				IF TriggerInput.Mode = TOUCHPROBEMODE_SINGLE_COMPATIBILITYMODE THEN
					CASE TriggerInput.Edge OF
						RisingEdge :
							IndexOffset := 16#201;
						FallingEdge:
							IndexOffset := 16#202;
					ELSE (* case *)
						Error := TRUE;
						ErrorID := MC_ERROR_INVALID_TOUCH_PROBE;
					END_CASE
				ELSE
					IF TcMcGlobal.NcDeviceInfoNcVersion > 16#020B07DD THEN
						IndexOffset := 16#200;  (* new from 2.11 NC driver 2014 *)
					ELSE
						(* new probe mode with old NC driver not possible *)
						Error := TRUE;
						ErrorID := MC_ERROR_INVALID_TOUCH_PROBE;
					END_IF
				END_IF

				IF TriggerInput.EncoderID > 255 THEN
					Error := TRUE;
					ErrorID := MC_ERROR_INVALID_TOUCH_PROBE;
				END_IF

				IF NOT Error THEN
					CASE TriggerInput.TouchProbe OF
						TouchProbe1,
						TouchProbe2,
						TouchProbe3,
						TouchProbe4:
							(* activate latch *)
							iTriggerInput := TriggerInput; (* save local copy *)
							ActTouchProbeActivate();
							iState := STATE_ORDER;

						PlcEvent:
							(* no action necessary here *);
							TriggerInput.ProbeState := TouchProbeActivated;
							iTriggerInput := TriggerInput; (* save local copy *)
							iState := STATE_WAITING;
					ELSE
						Error := TRUE;
						ErrorID := MC_ERROR_INVALID_TOUCH_PROBE;
					END_CASE
				END_IF
			END_IF
		END_IF

	STATE_ORDER :	(* wait until probe is activated *)
		ActTouchProbeActivate();

	STATE_WAITING : (* wait until touch probe was trigerred *)
		CASE iTriggerInput.TouchProbe OF (* type of touch probe *)
			TouchProbe1,
			TouchProbe2,
			TouchProbe3,
			TouchProbe4:
				IF TcMcGlobal.NcDeviceInfoNcVersion > 16#020B07DD AND stTouchProbeActivation.Mode<>INT_TO_UDINT(TOUCHPROBEMODE_SINGLE_COMPATIBILITYMODE) THEN
					(* new touch probe interface since TwinCAT 2.11 Nc-Driver 2014 *)
					ActTouchProbeMonitoring();
				ELSE
					(* classic touch probe interface until TwinCAT 2.11 Nc-Driver 2013 *)
					ActTouchProbeMonitorLatchValid();
					IF iState=STATE_WAITING THEN (* still not triggered *)
						ActTouchProbeMonitorActivity();
					END_IF
				END_IF

			(* CASE PlcEvent *)
			PlcEvent : (* touch proble will be triggered through a PLC signal (iTriggerInput.PlcEvent) *)
				ActTouchProbeMonitorPlcEvent();
		END_CASE (* type of touch probe *)

		IF NOT Done AND (TriggerInput.ProbeState = TouchProbeAborted) THEN
			(* function block has been aborted by an external MC_AbortTrigger *)
			CommandAborted := TRUE;
			iState := STATE_INITIALIZATION;
		END_IF

		IF TriggerInput.Mode = TOUCHPROBEMODE_CONTINOUS THEN
			(* check if probe triggered, then restart probe *)
			IF Done AND Execute THEN
(*				fbAdsReadState(READ:=FALSE); *)
(*				LastTouchProbeValue := TouchProbeValue;
				LastTouchProbeCounter := TouchProbeCounter;
				fbAdsReadLatchStatus(WRTRD:=TRUE); *)(* retrigger *)
				iState := STATE_WAITING; (* keep on waiting for next trigger *)
			ELSIF NOT Execute THEN (* abort trigger *)
				stTouchProbeDeactivation.TouchProbe := iTriggerInput.TouchProbe;
				stTouchProbeDeactivation.Edge := iTriggerInput.Edge;
				fbADSwrite(	WRITE:=FALSE); (* reset *)
				fbADSwrite(	NETID:= TcMcGlobal.NCNETID_TCMC,
							PORT:=AMSPORT_R0_NCSAF ,
							IDXGRP:=16#5200+TriggerInput.EncoderID ,
							IDXOFFS:=16#205,	(* deactivate touch probe *)
							LEN:= SIZEOF(stTouchProbeDeactivation),
							SRCADDR:=ADR(stTouchProbeDeactivation),
							WRITE:=TRUE ,
							TMOUT:=TcMcGlobal.tADSTimeOut);
				iState := 30000;
			END_IF
		END_IF

		IF iState<> STATE_WAITING THEN
			(* leave the waiting state now *)
			TriggerInput.ProbeState := TouchProbeInactive;
			fbAdsReadModulo(READ:=FALSE);	(* initialize again during next cycle *)
		END_IF

	30000 : (* abort trigger *)
		fbADSwrite();
		IF NOT fbAdsWrite.BUSY THEN
			IF fbAdsWrite.ERR THEN
				Error := fbAdsWrite.ERR;
				ErrorID := fbAdsWrite.ERRID;
			END_IF
			iState := STATE_INITIALIZATION;
		END_IF

END_CASE

ADSbusy := fbAdsWrite.BUSY OR fbAdsReadValid.BUSY OR fbAdsReadValue.BUSY OR fbAdsReadState.BUSY OR fbAdsReadModulo.BUSY;
IF iState=STATE_INITIALIZATION AND NOT Restart THEN
	(* reset Busy immediately  when sequence ends *)
	Busy := FALSE;
END_IF
END_FUNCTION_BLOCK
ACTION ActTouchProbeActivate:
(* start the touch probe sequence *)

(*LatchID := iTriggerInput.TouchProbe;*)
TriggerInput.ProbeState := TouchProbeActivated;
iTriggerInput.ProbeState := TouchProbeActivated;

(* read version of NC *)
(*
IF TcMcGlobal.NcDeviceInfoNcVersion=0 THEN
	TcMcGlobal.ReadDeviceInfo();
END_IF
*)

stTouchProbeActivation.TouchProbe := iTriggerInput.TouchProbe;
stTouchProbeActivation.Edge := iTriggerInput.Edge;
stTouchProbeActivation.Mode := iTriggerInput.Mode;
stTouchProbeActivation.SignalSource := iTriggerInput.SignalSource;	(* 20110218 KSt *)

IF stTouchProbeActivation.Mode = INT_TO_UDINT(TOUCHPROBEMODE_SINGLE_COMPATIBILITYMODE) THEN
	fbADSwrite(	NETID:= TcMcGlobal.NCNETID_TCMC,
				PORT:=AMSPORT_R0_NCSAF ,
				IDXGRP:=16#5200+iTriggerInput.EncoderID ,
				IDXOFFS:=IndexOffset,
				LEN:=0,
				SRCADDR:=ADR(stTouchProbeActivation),
				WRITE:=TRUE ,
				TMOUT:=TcMcGlobal.tADSTimeOut);
ELSE
	fbADSwrite(	NETID:= TcMcGlobal.NCNETID_TCMC,
				PORT:=AMSPORT_R0_NCSAF ,
				IDXGRP:=16#5200+iTriggerInput.EncoderID ,
				IDXOFFS:=IndexOffset,
				LEN:=SIZEOF(stTouchProbeActivation),
				SRCADDR:=ADR(stTouchProbeActivation),
				WRITE:=TRUE ,
				TMOUT:=TcMcGlobal.tADSTimeOut);
END_IF

IF NOT fbADSwrite.BUSY THEN
	IF fbADSwrite.ERR THEN
		Error := fbADSwrite.ERR;
		ErrorID := fbADSwrite.ERRID;
	END_IF
	IF NOT Error AND iTriggerInput.ProbeState = TouchProbeAborted THEN
		(* Synchronization error between MC_TouchProbe and MC_AbortTrigger *)
		Error := TRUE;
		ErrorID := MC_ERROR_TOUCH_PROBE_DEACTIVATED;
	END_IF
	iTriggerInput.ProbeState := SEL( Error, TouchProbeActivated, TouchProbeInactive );
	iState := SEL( Error, STATE_WAITING, STATE_INITIALIZATION);
END_IF
END_ACTION
ACTION ActTouchProbeMonitorActivity:
(* check if latch is still active *)
TimerAdsReadState(IN := NOT TimerAdsReadState.q , PT:=T#1s);
IF TimerAdsReadState.q OR fbAdsReadState.BUSY THEN
	fbAdsReadState(	NETID:= TcMcGlobal.NCNETID_TCMC,
				PORT:=AMSPORT_R0_NCSAF ,
				IDXGRP:=16#5100+TriggerInput.EncoderID ,
				IDXOFFS:= 16#201,
				LEN:= SIZEOF(TouchProbeActive[1]),
				DESTADDR:=ADR(TouchProbeActive) ,
				READ:=TRUE ,
				TMOUT:=TcMcGlobal.tADSTimeOut );
	IF NOT fbAdsReadState.BUSY THEN
		IF fbAdsReadState.ERR THEN
			Error := TRUE;
			ErrorID := fbAdsReadState.ERRID;
		ELSE
			IF TouchProbeActive[TriggerInput.TouchProbe]<>1 THEN
				TouchProbeInactiveCounter[TriggerInput.TouchProbe] := TouchProbeInactiveCounter[TriggerInput.TouchProbe] + 1;
				IF TouchProbeInactiveCounter[TriggerInput.TouchProbe] > 1 THEN
					(* error condition when the probing sequence is inactive more than once *)
					Error := TRUE;
					ErrorID := MC_ERROR_TOUCH_PROBE_DEACTIVATED;
					CommandAborted := TRUE;
					iState := STATE_INITIALIZATION;
				END_IF
			END_IF
		END_IF
		fbAdsReadState(READ:=FALSE); (* reset *)
	END_IF
END_IF
END_ACTION
ACTION ActTouchProbeMonitoring:
(* 	monitor if the touch probe has been triggered and if it is still active *)

(* 	new touch probe interface since 4/2010
	This action is only used with the new interface 
*)

Done := FALSE;		(* default *)
RecordedPosition := 0;	(* default *)

(* check if latch is still active and check for valid latch *)
TimerAdsReadState(IN := NOT TimerAdsReadState.q , PT:=T#1s);
IF ExternalLatchValid OR TimerAdsReadState.q OR fbAdsReadLatchStatus.BUSY THEN
	(* request for this probe unit *)
	stTouchProbeStatusRequest.TouchProbe := iTriggerInput.TouchProbe;

	fbAdsReadLatchStatus(
		NETID:= TcMcGlobal.NCNETID_TCMC,
		PORT:=AMSPORT_R0_NCSAF ,
		IDXGRP:=16#5100+iTriggerInput.EncoderID ,
		IDXOFFS:= 16#200,
		WRITELEN:= SIZEOF(stTouchProbeStatusRequest),
		READLEN:= SIZEOF(stTouchProbeStatusResponse),
		SRCADDR:= ADR(stTouchProbeStatusRequest),
		DESTADDR:= ADR(stTouchProbeStatusResponse),
		WRTRD:= TRUE,
		TMOUT:= TcMcGlobal.tADSTimeOut );

	IF NOT fbAdsReadLatchStatus.BUSY THEN
		IF fbAdsReadLatchStatus.ERR THEN
			Error := TRUE;
			ErrorID := fbAdsReadLatchStatus.ERRID;
		ELSE
			IF iTriggerInput.Edge = FallingEdge THEN
				TouchProbeActive[iTriggerInput.TouchProbe] := stTouchProbeStatusResponse.FallingEdgeActive;
				TouchProbeValid[iTriggerInput.TouchProbe] := stTouchProbeStatusResponse.FallingEdgeValid;
				TouchProbeValue[iTriggerInput.TouchProbe] := stTouchProbeStatusResponse.FallingEdgeValue;
				TouchProbeCounter[iTriggerInput.TouchProbe] := stTouchProbeStatusResponse.FallingEdgeCounter;
			ELSE
				TouchProbeActive[iTriggerInput.TouchProbe] := stTouchProbeStatusResponse.RisingEdgeActive;
				TouchProbeValid[iTriggerInput.TouchProbe] := stTouchProbeStatusResponse.RisingEdgeValid;
				TouchProbeValue[iTriggerInput.TouchProbe] := stTouchProbeStatusResponse.RisingEdgeValue;
				TouchProbeCounter[iTriggerInput.TouchProbe] := stTouchProbeStatusResponse.RisingEdgeCounter;
			END_IF
			IF TouchProbeValid[iTriggerInput.TouchProbe] = 1 THEN
				IF  iTriggerInput.Mode <> TOUCHPROBEMODE_CONTINOUS		(* single mode *)
					OR LastTouchProbeValue[ iTriggerInput.TouchProbe ] <> TouchProbeValue[ iTriggerInput.TouchProbe ] 	(* or continous mode and value changed *)
					OR LastTouchProbeCounter[ iTriggerInput.TouchProbe ] <> TouchProbeCounter[ iTriggerInput.TouchProbe ](* or continous mode and counter changed *)
					THEN (* new position recorded  *)
					RecordedPosition:=TouchProbeValue[iTriggerInput.TouchProbe];
					LastTouchProbeValue := TouchProbeValue;
					LastTouchProbeCounter := TouchProbeCounter;
					Done := TRUE;
					IF TriggerInput.ModuloPositions AND (ModuloFactor<>0) THEN	(* check for  (ModuloFactor=0) - 2007-02-06 KSt *)
						RecordedPosition := MODABS(RecordedPosition,  ModuloFactor);
						TouchProbeModuloValue[TriggerInput.TouchProbe] := RecordedPosition;
(*						InWindow := (RecordedPosition>=FirstPosition) AND (RecordedPosition<=LastPosition);*)	(* 20110216 KSt *)
						IF FirstPosition>LastPosition THEN (* 20110216 KSt *)
							InWindow := (RecordedPosition>=FirstPosition) OR  (RecordedPosition<=LastPosition);  (* 20110216 KSt *)
						ELSE
							InWindow := (RecordedPosition>=FirstPosition) AND (RecordedPosition<=LastPosition);
						END_IF
					ELSE
						InWindow := (RecordedPosition>=FirstPosition) AND (RecordedPosition<=LastPosition);
					END_IF
					IF WindowOnly AND NOT InWindow THEN
						RecordedPosition:=0;
						Done := FALSE;
						Restart := TRUE; (* ignore this event, latch next one *)
					ELSE
						(* fill RecordedData structure *)
						RecordedData.RecordedPosition := RecordedPosition;
						RecordedData.Counter:=TouchProbeCounter[TriggerInput.TouchProbe];
						RecordedData.AbsolutePosition := TouchProbeValue[iTriggerInput.TouchProbe];
						IF ModuloFactor = 0 THEN
							RecordedData.ModuloPosition := MODABS(RecordedData.AbsolutePosition,  360);
						ELSE
							RecordedData.ModuloPosition := MODABS(RecordedData.AbsolutePosition,  ModuloFactor);
						END_IF
					END_IF
					iState := STATE_INITIALIZATION;
				END_IF
			ELSIF TouchProbeActive[iTriggerInput.TouchProbe] <> 1 THEN
				TouchProbeInactiveCounter[iTriggerInput.TouchProbe] := TouchProbeInactiveCounter[iTriggerInput.TouchProbe] + 1;
				IF TouchProbeInactiveCounter[iTriggerInput.TouchProbe] > 1 THEN
					(* error condition when the probing sequence is inactive more than once *)
					Error := TRUE;
					ErrorID := MC_ERROR_TOUCH_PROBE_DEACTIVATED;
					CommandAborted := TRUE;
					iState := STATE_INITIALIZATION;
				END_IF
			END_IF
		END_IF
		fbAdsReadLatchStatus(WRTRD:=FALSE); (* reset *)
		IF iTriggerInput.Mode=TOUCHPROBEMODE_CONTINOUS AND Execute THEN
			fbAdsReadLatchStatus(WRTRD:=TRUE); (* retrigger *)
		END_IF
	END_IF
END_IF
END_ACTION
ACTION ActTouchProbeMonitorLatchValid:
(* monitor if the touch probe has been triggered *)

IF F_AxisExternalLatchValid(Axis.NcToPlc.StateDWord) THEN
	(* read the status of the latch *)
	fbAdsReadValid(	NETID:= TcMcGlobal.NCNETID_TCMC,
				PORT:=AMSPORT_R0_NCSAF ,
				IDXGRP:=16#5100+TriggerInput.EncoderID ,
				IDXOFFS:= 16#202,
				LEN:= SIZEOF(TouchProbeValid[1]),
				DESTADDR:=ADR(TouchProbeValid) ,
				READ:=TRUE ,
				TMOUT:=TcMcGlobal.tADSTimeOut );
	(* read the latched value *)
	fbAdsReadValue(	NETID:= TcMcGlobal.NCNETID_TCMC,
				PORT:=AMSPORT_R0_NCSAF ,
				IDXGRP:=16#5100+TriggerInput.EncoderID ,
				IDXOFFS:= 16#205,
				LEN:=SIZEOF(TouchProbeValue[1]),
				DESTADDR:=ADR(TouchProbeValue) ,
				READ:=TRUE ,
				TMOUT:=TcMcGlobal.tADSTimeOut );
	IF NOT fbAdsReadValid.BUSY AND NOT fbAdsReadValue.BUSY THEN
		IF fbAdsReadValid.err THEN
			Error := TRUE;
			ErrorID := fbAdsReadValid.ERRID;
			iState := STATE_INITIALIZATION;
		ELSIF fbAdsReadValue.err THEN
			Error := TRUE;
			ErrorID := fbAdsReadValue.ERRID;
			iState := STATE_INITIALIZATION;
		ELSE (* no error *)
			IF TouchProbeValid[TriggerInput.TouchProbe]=1 THEN
				RecordedPosition:=TouchProbeValue[TriggerInput.TouchProbe];
				Done := TRUE;
				IF TriggerInput.ModuloPositions AND (ModuloFactor<>0) THEN	(* check for  (ModuloFactor=0) - 2007-02-06 KSt *)
					RecordedPosition := MODABS(RecordedPosition,  ModuloFactor);
					TouchProbeModuloValue[TriggerInput.TouchProbe] := RecordedPosition;
(*					InWindow := (RecordedPosition>=FirstPosition) AND (RecordedPosition<=LastPosition);*)  (* 20110216 KSt *)
					IF FirstPosition>LastPosition THEN (* 20110216 KSt *)
						InWindow := (RecordedPosition>=FirstPosition) OR  (RecordedPosition<=LastPosition);  (* 20110216 KSt *)
					ELSE
						InWindow := (RecordedPosition>=FirstPosition) AND (RecordedPosition<=LastPosition);
					END_IF
				ELSE
					InWindow := (RecordedPosition>=FirstPosition) AND (RecordedPosition<=LastPosition);
				END_IF
				IF WindowOnly AND NOT InWindow THEN
					RecordedPosition:=0;
					Done := FALSE;
					Restart := TRUE; (* ignore this event, latch next one *)
				ELSE
					(* fill RecordedData structure *)
					RecordedData.RecordedPosition := RecordedPosition;
					RecordedData.Counter:=TouchProbeCounter[TriggerInput.TouchProbe];
					RecordedData.AbsolutePosition := TouchProbeValue[TriggerInput.TouchProbe];
					IF ModuloFactor = 0 THEN
						RecordedData.ModuloPosition := MODABS(RecordedData.AbsolutePosition,  360);
					ELSE
						RecordedData.ModuloPosition := MODABS(RecordedData.AbsolutePosition,  ModuloFactor);
					END_IF
				END_IF
				iState := STATE_INITIALIZATION;
			ELSE
				fbAdsReadValid(READ:=FALSE);
				fbAdsReadValue(READ:=FALSE);
			END_IF
		END_IF
	END_IF
END_IF
END_ACTION
ACTION ActTouchProbeMonitorPlcEvent:
(* touch probe sequence for simple PLC inputs *)
(* monitor PLC input trigger *)

RtrigPlcEvent(CLK:=TriggerInput.PlcEvent);
FtrigPlcEvent(CLK:=TriggerInput.PlcEvent);
IF ((TriggerInput.Edge=RisingEdge) AND RtrigPlcEvent.Q) OR
   ((TriggerInput.Edge=FallingEdge) AND FtrigPlcEvent.Q) THEN
	RecordedPosition:=Axis.NcToPlc.ActPos; 	(* 2007-02-06 KSt *)
	IF TriggerInput.ModuloPositions AND (ModuloFactor<>0) THEN	(* check for  (ModuloFactor=0) - 2007-02-06 KSt *)
		RecordedPosition :=  MODABS(RecordedPosition,  ModuloFactor);
(*		InWindow := (RecordedPosition>=FirstPosition) AND (RecordedPosition<=LastPosition);*)  (* 20110216 KSt *)
		IF FirstPosition>LastPosition THEN (* 20110216 KSt *)
			InWindow := (RecordedPosition>=FirstPosition) OR  (RecordedPosition<=LastPosition);  (* 20110216 KSt *)
		ELSE
			InWindow := (RecordedPosition>=FirstPosition) AND (RecordedPosition<=LastPosition);
		END_IF
	ELSE
		InWindow := (RecordedPosition>=FirstPosition) AND (RecordedPosition<=LastPosition);
	END_IF
	IF WindowOnly AND NOT InWindow THEN
		RecordedPosition:=0;	(* 2007-02-06 KSt *)
	ELSE
		(* fill RecordedData structure *)
		RecordedData.RecordedPosition := RecordedPosition;
		RecordedData.Counter := RecordedData.Counter + 1;
		RecordedData.AbsolutePosition := Axis.NcToPlc.ActPos;
		IF ModuloFactor = 0 THEN
			RecordedData.ModuloPosition := MODABS(RecordedData.AbsolutePosition,  360);
		ELSE
			RecordedData.ModuloPosition := MODABS(RecordedData.AbsolutePosition,  ModuloFactor);
		END_IF
		Done := TRUE;
		iState := STATE_INITIALIZATION;
	END_IF
END_IF
END_ACTION
ACTION ActTouchProbeStartupInit:
(* initialization on plc start-up *)
(* read the axis' modulo factor *)

IF TriggerInput.ModuloPositions THEN
	IF ModuloFactor = 0 THEN
		InitDone := FALSE; (* 2007-02-06 KSt *)
	END_IF
	fbAdsReadModulo(	NETID:= TcMcGlobal.NCNETID_TCMC,
						PORT:= AMSPORT_R0_NCSAF,
						IDXGRP:= 16#5000+TriggerInput.EncoderID ,
						IDXOFFS:= 16#9,
						LEN:= SIZEOF(ModuloFactor),
						DESTADDR:= ADR(ModuloFactor),
						READ:= TRUE,
						TMOUT:= TcMcGlobal.tADSTimeOut);
	IF NOT fbAdsReadModulo.BUSY THEN
		IF fbAdsReadModulo.ERR OR (ModuloFactor=0) THEN
			fbAdsReadModulo( READ:=FALSE ); 	(* 2007-02-06 KSt *)
			InitDone := FALSE; 	(* init failed - 2007-02-06 KSt *)
			Error := TRUE;
			ErrorID := fbAdsReadModulo.ERRID;
		ELSE
			InitDone := TRUE;
		END_IF
	END_IF
ELSE (* no modulo positions *)
	fbAdsReadModulo( READ:=FALSE );	(* 2007-02-06 KSt *)
	InitDone := TRUE;
END_IF
END_ACTION

(* POU MC_WriteBoolParameter, ST *)
FUNCTION_BLOCK MC_WriteBoolParameter
(*	This Function Block modifies the value of a vendor specific boolean parameter. *)
VAR_IN_OUT
	Axis				:	AXIS_REF;	(* B *)
END_VAR
VAR_INPUT
	Execute			:	BOOL;	(* B *)
	ParameterNumber	:	INT;		(* B *)
	Value			:	BOOL;	(* B *)
(* 	ExecutionMode 	: 	MC_EXECUTION_MODE *)	(* E *)	(* not available *)
END_VAR
VAR_OUTPUT
	Done			:	BOOL;	(* B *)
	Busy			: 	BOOL;	(* E *)
	Error			:	BOOL;	(* B *)
	ErrorID			:	UDINT;	(* E *)
END_VAR
VAR
	ADSbusy		: 	BOOL;
	fbReadWriteParameter: 	_FB_ReadWriteParameter;
END_VAR
{library private}
VAR
	nParatype 		:	_E_ParameterType;
	dwValue 			: 	DWORD;
	lrValue 			: 	LREAL;
	fbTrigger 		: 	R_TRIG;
END_VAR
IF NOT Execute THEN
	Done := FALSE;
	Error := FALSE;			(* reset at falling edge of Execute *)
	ErrorID := 0;
END_IF
fbTrigger(CLK:= Execute);
IF fbTrigger.Q AND NOT Busy THEN
	Busy := TRUE;
	Done := FALSE;
	Error := FALSE;
	ErrorID := MC_ERROR_NO_ERROR;
END_IF;
(* *)
IF Busy THEN
	nParatype := PARAMETERTYPE_BOOL;
	fbReadWriteParameter(Enable:= TRUE, ParameterNumber:= ParameterNumber, Mode:= READWRITEPARAMETERMODE_WRITE,
						ParameterType:=nParatype, Axis:= Axis, ValueLreal:= lrValue, ValueDword := dwValue, ValueBool := Value);
	IF fbReadWriteParameter.Done THEN
		Done := TRUE;
		Busy := FALSE;
		fbReadWriteParameter(Enable:= FALSE, ParameterNumber:= ParameterNumber, Mode:= READWRITEPARAMETERMODE_WRITE,
						ParameterType:= nParatype , Axis:= Axis, ValueLreal:= lrValue, ValueDword := dwValue, ValueBool := Value);
	END_IF;
	IF fbReadWriteParameter.Error THEN
		Busy := FALSE;
		Done := FALSE;
		Error := TRUE;
		ErrorID := fbReadWriteParameter.ErrorID;
		fbReadWriteParameter(Enable:= FALSE, ParameterNumber:= ParameterNumber, Mode:= READWRITEPARAMETERMODE_WRITE,
						ParameterType:= nParatype , Axis:= Axis, ValueLreal:= lrValue, ValueDword := dwValue, ValueBool := Value);
	END_IF;
END_IF;

ADSbusy := fbReadWriteParameter.ADSbusy;
END_FUNCTION_BLOCK

(* POU MC_WriteParameter, ST *)
FUNCTION_BLOCK MC_WriteParameter
(*	This Function Block modifies the value of a vendor specific parameter. *)
VAR_IN_OUT
	Axis				:	AXIS_REF;	(* B *)
END_VAR
VAR_INPUT
	Execute			:	BOOL;		(* B *)
	ParameterNumber	:	INT;			(* B *)
	Value			:	LREAL;		(* B *)
(* 	ExecutionMode 	: 	MC_EXECUTION_MODE *)	(* E *)	(* not available *)
END_VAR
VAR_OUTPUT
	Done			:	BOOL;		(* B *)
	Busy			: 	BOOL;		(* E *)
	Error			:	BOOL;		(* B *)
	ErrorID			:	UDINT;		(* E *)
END_VAR
VAR
	ADSbusy		: 	BOOL;
	fbReadWriteParameter: _FB_ReadWriteParameter;
END_VAR
{library private}
VAR
	nParatype 		:	_E_ParameterType;
	dwValue 			: 	DWORD;
	bValue 			: 	BOOL;
	fbTrigger 		: 	R_TRIG;
END_VAR
IF NOT Execute THEN
	Done := FALSE;
	Error := FALSE;			(* reset at falling edge of Execute *)
	ErrorID := 0;
END_IF
fbTrigger(CLK:= Execute);
IF fbTrigger.Q AND NOT Busy THEN
	Busy := TRUE;
	Done := FALSE;
	Error := FALSE;
	ErrorID := MC_ERROR_NO_ERROR;
END_IF;
(* *)
IF Busy THEN
	nParatype := PARAMETERTYPE_LREAL;
	bValue := Value<>0; (* 2010-05-04 KST - to write bool parameters with MC_WriteParameter as well *)
	fbReadWriteParameter(Enable:= TRUE, ParameterNumber:= ParameterNumber, Mode:= READWRITEPARAMETERMODE_WRITE,
						ParameterType:=nParatype, Axis:= Axis, ValueLreal:= Value, ValueDword := dwValue, ValueBool := bValue);
	IF fbReadWriteParameter.Done THEN
		Done := TRUE;
		Busy := FALSE;
		fbReadWriteParameter(Enable:= FALSE, ParameterNumber:= ParameterNumber, Mode:= READWRITEPARAMETERMODE_WRITE,
						ParameterType:= nParatype , Axis:= Axis, ValueLreal:= Value, ValueDword := dwValue, ValueBool := bValue);
	END_IF;
	IF fbReadWriteParameter.Error THEN
		Busy := FALSE;
		Done := FALSE;
		Error := TRUE;
		ErrorID := fbReadWriteParameter.ErrorID;
		fbReadWriteParameter(Enable:= FALSE, ParameterNumber:= ParameterNumber, Mode:= READWRITEPARAMETERMODE_WRITE,
						ParameterType:= nParatype , Axis:= Axis, ValueLreal:= Value, ValueDword := dwValue, ValueBool := bValue);
	END_IF;
END_IF;

ADSbusy := fbReadWriteParameter.ADSbusy;
END_FUNCTION_BLOCK
